(*
A DWORD alias type to be used with PLC HMI. Encodes ARGB value.
*)
TYPE Argb : DWORD; END_TYPE

(* stored: Version 1.1.0.1
   DUT Argb: Id {8a6bcbc4-7e62-43a0-b446-48bdd11ecd5a} *)
